{attribute addProperty BoxType "EJ2522-0000-0022"}
{attribute addProperty Id "Set_counterBIT10.1253ReservedBIT10.12516"}
{attribute addProperty CRC "2811377587"}
{attribute addProperty SizeInBites "16"}
{attribute addProperty SizeInBytes "2"}
TYPE Control_A79237B3 :
STRUCT
	{attribute 'hide'}
	reserve_1_BIT_0 : BOOL;
	{attribute 'hide'}
	reserve_1_BIT_1 : BOOL;
	{attribute addProperty Name "Set_counter"}
	Set_counter : BOOL;
	{attribute 'hide'}
	reserve_2_BIT_0 : BOOL;
	{attribute 'hide'}
	reserve_2_BIT_1 : BOOL;
	{attribute 'hide'}
	reserve_2_BIT_2 : BOOL;
	{attribute 'hide'}
	reserve_2_BIT_3 : BOOL;
	{attribute 'hide'}
	reserve_2_BIT_4 : BOOL;
	{attribute 'hide'}
	reserve_2_BIT_5 : BOOL;
	{attribute 'hide'}
	reserve_2_BIT_6 : BOOL;
	{attribute 'hide'}
	reserve_2_BIT_7 : BOOL;
	{attribute 'hide'}
	reserve_2_BIT_8 : BOOL;
	{attribute 'hide'}
	reserve_2_BIT_9 : BOOL;
	{attribute 'hide'}
	reserve_2_BIT_10 : BOOL;
	{attribute 'hide'}
	reserve_2_BIT_11 : BOOL;
	{attribute addProperty Name "Reserved"}
	Reserved : BOOL;
END_STRUCT
END_TYPE

(* stored: Version 1.2.0.0, ProductVersion 3.1.4024.9
   DUT Control_A79237B3: Id {7ee0d042-910d-40cb-b757-fd26e2f1dc1c} *)
